Staubli VAL3: PA_grinding_V3.pjx

--- PA_grinding_V3.pjx ---
Parameters version=s7.11.2 stackSize=5000 millimeterUnit=true
Program file=start.pgx
Program file=stop.pgx
Program file=_mainLoop.pgx
Program file=_moveToScan.pgx
Program file=_recvWaypoints.pgx
Program file=_recvFloat.pgx
Program file=_sendStatus.pgx
Program file=_startPass.pgx
Program file=_finish.pgx
Data file=PA_grinding_V3.dtx

--- PA_grinding_V3.dtx ---
public tool tTool = {z=100, fatherId=flange[0], ioLink=valve1}
public frame fWork = {fatherId=world[0]}
public jointRx j_home = {j1=83.61, j2=38.15, j3=96.24, j4=-4.09, j5=-58.18, j6=-4.12}
public jointRx j_scan = {j1=83.61, j2=38.15, j3=96.24, j4=-4.09, j5=-58.18, j6=-4.12}
public jointRx jWaypoints[100]
public num nWaypointCount
public num nForceTarget
public num nDOC
public num nCmdSignal
public num nStatusSignal
num nLastCmd
bool bRunning
num i
mdesc mNomSpeed = {tmax=200, rmax=200, blend=off}
mdesc mGrindSpeed = {tmax=30, rmax=30, leave=1, reach=1, blend=off}
public sio siTcpIpCommand = {link=Socket\Command}
public sio siTcpIpMotion = {link=Socket\Motion}
public sio siTcpIpFbk = {link=Socket\Feedback}
public num nConnFlag
num nByte
public pointRx curent_pos = {fatherId=world[0]}
mdesc mAprSpeed = {tmax=5, rmax=5, blend=off}
public aio aiECAT1_0 = {link=EtherCAT-1\%IF0}
public aio aoECAT1_0 = {link=EtherCAT-1\%QF0}
public aio aoECAT1_32 = {link=EtherCAT-1\%QF32}
public aio aoECAT1_64 = {link=EtherCAT-1\%QF64}
public aio aoECAT1_96 = {link=EtherCAT-1\%QF96}
public aio aoECAT1_128 = {link=EtherCAT-1\%QF128}
public aio aoECAT1_160 = {link=EtherCAT-1\%QF160}

--- start.pgx ---
program start()
begin
  // ============================================================================
  // PA_grinding_V3 - TCP 통신 버전 (3 소켓)
  // Command (11001): ROS2 -> 로봇, 명령 수신
  // Motion (11000): ROS2 -> 로봇, Waypoint/Joint 데이터
  // Feedback (11002): 로봇 -> ROS2, 상태 송신
  // ============================================================================

  userPage()
  cls()
  putln("=================================")
  putln("  PA_grinding_V3 Started")
  putln("=================================")
  putln("")

  // 초기화
  bRunning = true
  nLastCmd = 0
  nStatusSignal = 0
  nWaypointCount = 0
  nConnFlag = 0

  // 소켓 타임아웃 설정 (non-blocking)
  sioCtrl(siTcpIpCommand, "timeout", 0)
  sioCtrl(siTcpIpMotion, "timeout", 0)
  sioCtrl(siTcpIpFbk, "timeout", 0)

  // 버퍼 클리어
  clearBuffer(siTcpIpCommand)
  clearBuffer(siTcpIpMotion)
  clearBuffer(siTcpIpFbk)

  putln("TCP 소켓 준비 완료")
  putln("  - Command: 11001 (수신)")
  putln("  - Motion: 11000 (수신)")
  putln("  - Feedback: 11002 (송신)")
  putln("")
  putln("명령 대기 중...")
  putln("CMD: 1=종료, 2=스캔이동, 3=WP수신, 4=가공")
  putln("")

  // 메인 루프 태스크 시작
  taskCreate "mainLoop", 100, _mainLoop()

  // 메인 루프 종료 대기
  wait(taskStatus("mainLoop") == -1)

  cls()
  putln("PA_grinding_V3 종료됨")

end

--- _finish.pgx ---
program _finish()
begin
  // ============================================================================
  // CMD 1: 종료 - 홈 위치 복귀
  // ============================================================================
  cls()
  putln("[CMD 1] 종료 - 홈 복귀")
  nStatusSignal = 0

  movej(j_home, tTool, mNomSpeed)
  waitEndMove()

  putln("[CMD 1] 완료")
  bRunning = false

end

--- _mainLoop.pgx ---
program _mainLoop()
  local num l_nRetVal
begin
  // ============================================================================
  // 메인 루프 - Command 소켓에서 명령 수신
  // 명령: 1바이트 (1=종료, 2=스캔, 3=WP수신, 4=가공)
  // ============================================================================

  while bRunning

    // Command 소켓에서 명령 수신 (1바이트)
    l_nRetVal = sioGet(siTcpIpCommand, nByte)

    if l_nRetVal == 1
      // 데이터 수신됨
      nCmdSignal = nByte
      nConnFlag = 1
      putln("[CMD] 수신 = " + toString("", nCmdSignal))

      switch nCmdSignal
        case 1
          call _finish()
          break
        case 2
          call _moveToScan()
          break
        case 3
          call _recvWaypoints()
          break
        case 4
          call _startPass()
          break
        default
          putln("[WARN] 알 수 없는 명령: " + toString("", nCmdSignal))
          break
      endSwitch

      // Feedback 소켓으로 상태 응답 전송
      call _sendStatus()

    elseIf l_nRetVal == -1
      // 연결 끊김
      if nConnFlag == 1
        putln("[CMD] 연결 끊김")
        nConnFlag = 0
      endIf
    endIf

    delay(0.01)

  endWhile

end

--- _moveToScan.pgx ---
program _moveToScan()
begin
  // ============================================================================
  // CMD 2: 스캔 위치로 이동
  // ============================================================================
  cls()
  putln("[CMD "+ toString("", nCmdSignal) +"] 스캔 위치로 이동")
  nStatusSignal = 0

  movej(j_scan, tTool, mNomSpeed)
  waitEndMove()

  putln("[CMD 2] 완료 - STATUS=1")
  nStatusSignal = 1

end

--- _recvFloat.pgx ---
program _recvFloat(num& x_nValue)
  local num l_nRetVal
  local num l_nBytes[4]
  local num l_nCount
  local num l_nByte
  local num l_nSign
  local num l_nExp
  local num l_nMant
begin
  // ============================================================================
  // IEEE 754 float32 수신 및 파싱 (little-endian)
  // ============================================================================

  // 4바이트 수신
  l_nCount = 0
  while l_nCount < 4
    l_nRetVal = sioGet(siTcpIpMotion, l_nByte)
    if l_nRetVal == 1
      l_nBytes[l_nCount] = l_nByte
      l_nCount = l_nCount + 1
    elseIf l_nRetVal == -1
      x_nValue = 0
      return
    endIf
  endWhile

  // IEEE 754 float32 파싱 (little-endian)
  l_nSign = roundDown(l_nBytes[3] / 128)
  l_nExp = (l_nBytes[3] - l_nSign * 128) * 2 + roundDown(l_nBytes[2] / 128)
  l_nMant = (l_nBytes[2] - roundDown(l_nBytes[2] / 128) * 128) * 65536 + l_nBytes[1] * 256 + l_nBytes[0]

  if l_nExp == 0
    x_nValue = 0
  elseIf l_nExp == 255
    x_nValue = 0
  else
    x_nValue = power(2, l_nExp - 127) * (1 + l_nMant / 8388608)
    if l_nSign == 1
      x_nValue = -x_nValue
    endIf
  endIf

end

--- _recvWaypoints.pgx ---
program _recvWaypoints()
  local num l_nJ1
  local num l_nJ2
  local num l_nJ3
  local num l_nJ4
  local num l_nJ5
  local num l_nJ6
begin
  // ============================================================================
  // CMD 3: 웨이포인트 수신 (TCP - Motion 소켓)
  // 데이터: DOC(float) + Force(float) + Count(float) + Joints(6 floats each)
  // Joint: j1, j2, j3, j4, j5, j6 (degrees)
  // ============================================================================
  cls()
  putln("[CMD "+ toString("", nCmdSignal) +"] 웨이포인트 수신 시작")
  nStatusSignal = 0

  // DOC 수신
  call _recvFloat(nDOC)

  // Force 수신
  call _recvFloat(nForceTarget)

  // Count 수신
  call _recvFloat(nWaypointCount)
  nWaypointCount = roundDown(nWaypointCount)

  putln("  DOC=" + toString("", nDOC))
  putln("  Force=" + toString("", nForceTarget))
  putln("  Count=" + toString("", nWaypointCount))

  // 각 Waypoint 수신 (6축 Joint)
  for i = 0 to nWaypointCount - 1
    call _recvFloat(l_nJ1)
    call _recvFloat(l_nJ2)
    call _recvFloat(l_nJ3)
    call _recvFloat(l_nJ4)
    call _recvFloat(l_nJ5)
    call _recvFloat(l_nJ6)

    jWaypoints[i].j1 = l_nJ1
    jWaypoints[i].j2 = l_nJ2
    jWaypoints[i].j3 = l_nJ3
    jWaypoints[i].j4 = l_nJ4
    jWaypoints[i].j5 = l_nJ5
    jWaypoints[i].j6 = l_nJ6

    putln("  J[" + toString("", i) + "]=" + toString("", l_nJ1) + "," + toString("", l_nJ2) + "," + toString("", l_nJ3) + "," + toString("", l_nJ4) + "," + toString("", l_nJ5) + "," + toString("", l_nJ6))
  endFor

  putln("[CMD 3] 완료")
  nStatusSignal = 3

end

--- _sendStatus.pgx ---
program _sendStatus()
  local num l_nData
begin
  // ============================================================================
  // 상태 응답 전송 (1바이트)
  // 0=Idle, 1=Ready, 2=PassDone, 3=Error
  // ============================================================================

  l_nData = nStatusSignal
  sioSet(siTcpIpFbk, l_nData)
  putln("[TCP] STATUS = " + toString("", nStatusSignal))

end

--- _startPass.pgx ---
program _startPass()
  local pointRx l_pStart
  local pointRx l_pEnd
  local pointRx l_pApproach
  local pointRx l_pRetract
  local num l_nHeight
begin
  // ============================================================================
  // CMD 4: 그라인딩 패스 실행
  // 1. 시작점 위 (Approach) 이동
  // 2. 시작점 이동
  // 3. 웨이포인트 순차 이동 (가공)
  // 4. 끝점 위 (Retract) 이동
  // ============================================================================
  cls()
  putln("[CMD "+ toString("", nCmdSignal) +"] 가공 시작")
  putln("  Waypoints: " + toString("", nWaypointCount))
  putln("  DOC: " + toString("", nDOC))
  putln("  Force: " + toString("", nForceTarget))
  nStatusSignal = 0

  if nWaypointCount <= 0
    putln("[ERROR] 웨이포인트 없음")
    nStatusSignal = 3
    return
  endIf

  // Approach/Retract 높이 설정 (mm)
  l_nHeight = 10

  // 시작점, 끝점의 직교좌표 계산
  l_pStart = jointToPoint(tTool, fWork, jWaypoints[0])
  l_pEnd = jointToPoint(tTool, fWork, jWaypoints[nWaypointCount - 1])

  // Approach 포인트 (시작점 위)
  l_pApproach = l_pStart
  l_pApproach.trsf.z = l_pApproach.trsf.z + l_nHeight

  // Retract 포인트 (끝점 위)
  l_pRetract = l_pEnd
  l_pRetract.trsf.z = l_pRetract.trsf.z + l_nHeight

  // 1. Approach 위치로 이동
  putln("  [1] Approach 이동 (Z+" + toString("", l_nHeight) + ")")
  movel(l_pApproach, tTool, mNomSpeed)
  waitEndMove()

  // 2. 시작점으로 하강
  putln("  [2] 시작점 하강")
  movel(l_pStart, tTool, mAprSpeed)
  waitEndMove()

  // 3. 가공 경로 실행
  cls()
  putln("  [CMD 4] 가공 경로 실행")
  for i = 0 to nWaypointCount - 1
    putln("    -> WP[" + toString("", i) + "]")
    movej(jWaypoints[i], tTool, mGrindSpeed)
    waitEndMove()
    // TODO: Force Control 적용
  endFor

  // 4. Retract 위치로 상승
  putln("  [4] Retract 이동 (Z+" + toString("", l_nHeight) + ")")
  movel(l_pRetract, tTool, mAprSpeed)
  waitEndMove()

  movej(j_scan, tTool, mNomSpeed)
  waitEndMove()

  nStatusSignal = 4
  putln("[CMD 4] 완료 - STATUS=4")


end

--- stop.pgx ---
program stop()
begin
  bRunning = false
  taskKill("mainLoop")
end
